FUNCTION_BLOCK FB_Clamp_INT_Test  EXTENDS TcUnit.FB_TestSuite

OutOfBoundsUpper();
OutOfBoundsLower();
ValidInput();

METHOD OutOfBoundsLower : REFERENCE TO FB_Test
VAR
	Input : INT := -100;
	Upper : INT := 180;
	Lower : INT := 0;
	ExpectedOutput : INT := 0;
	ActualOutput : INT;
	Clamp: FB_Clamp_INT;
END_VAR
TEST('TEST: Out of bounds lower');

Clamp(
	Input:= Input, 
	UpperLimit:= Upper, 
	LowerLimit:= Lower, 
	Output=> ActualOutput, 
	OutOfBounds=> );

	
AssertEquals(Expected := ExpectedOutput,
	Actual := ActualOutput,
	Message := 'Not expected output');

TEST_FINISHED();
END_METHOD

METHOD OutOfBoundsUpper
VAR
	Input : INT := 200;
	Upper : INT := 180;
	Lower : INT := 0;
	ExpectedOutput : INT := 180;
	ActualOutput : INT;
	Clamp: FB_Clamp_INT;
END_VAR
TEST('TEST: Out of bounds upper');

Clamp(
	Input:= Input, 
	UpperLimit:= Upper, 
	LowerLimit:= Lower, 
	Output=> ActualOutput, 
	OutOfBounds=> );

	
AssertEquals(Expected := ExpectedOutput,
	Actual := ActualOutput,
	Message := 'Not expected output');

TEST_FINISHED();
END_METHOD

METHOD ValidInput
VAR
	Input : INT := 150;
	Upper : INT := 180;
	Lower : INT := 0;
	ExpectedOutput : INT := 150;
	ActualOutput : INT;
	Clamp: FB_Clamp_INT;
END_VAR
TEST('TEST: Valid input');

Clamp(
	Input:= Input, 
	UpperLimit:= Upper, 
	LowerLimit:= Lower, 
	Output=> ActualOutput, 
	OutOfBounds=> );

	
AssertEquals(Expected := ExpectedOutput,
	Actual := ActualOutput,
	Message := 'Not expected output');

TEST_FINISHED();
END_METHOD

END_FUNCTION_BLOCK

(* stored: Version 1.1.0.1, ProductVersion 3.1.4024.13
   POU FB_Clamp_INT_Test: Id {75fcef52-5ac9-4e10-ba14-518f6b1b3301}, SpecialFunc None
   Method OutOfBoundsLower: Id {536cf890-3896-4b8f-b0f3-3fc4db3dbc65}
   Method OutOfBoundsUpper: Id {0d02038d-9e4f-4be6-8898-4127215ba0b4}
   Method ValidInput: Id {d6dba15a-9e40-44eb-a58b-29f170bdc2b3} *)
